// LS Electric XG5000 project: 2016-46
// PLC NewPLC
// module base 0 slot 0: 입출력 모듈:XBC-DR20E (DC 24V 입력 12점, 릴레이 출력 8점)

PROGRAM NewProgram (task: 스캔 프로그램)

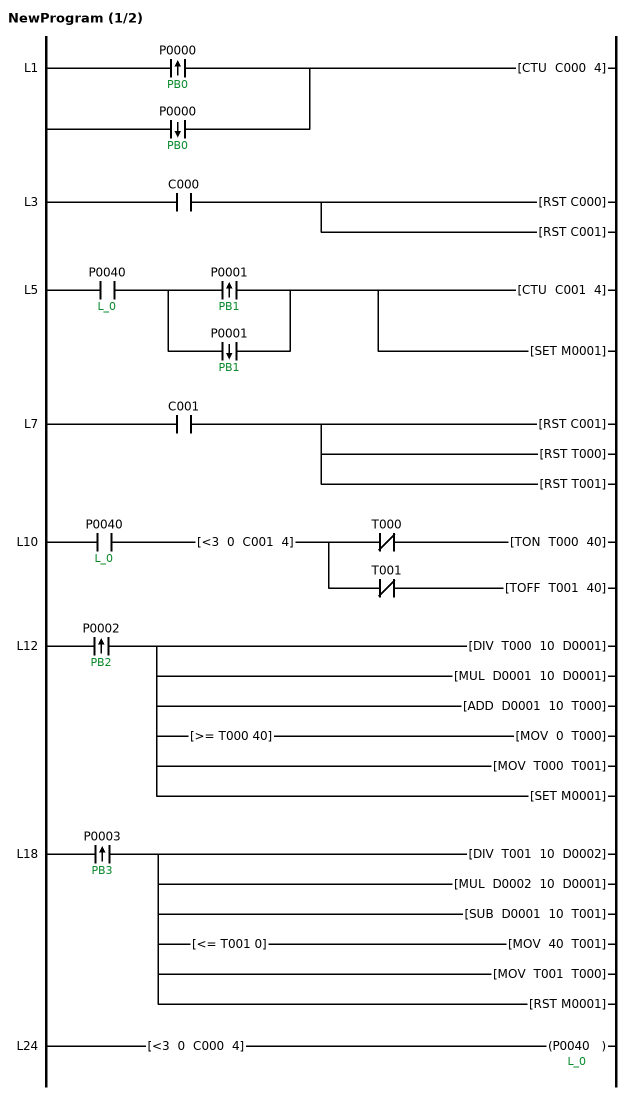
; L1
LOADP     P0000	// PB0
ORN       P0000	// PB0
CTU       C000 4
; L3
LOAD      C000
RST       C000
RST       C001
; L5
LOAD      P0040	// L_0
LOADP     P0001	// PB1
ORN       P0001	// PB1
AND LOAD
CTU       C001 4
SET       M0001
; L7
LOAD      C001
RST       C001
RST       T000
RST       T001
; L10
LOAD      P0040	// L_0
AND<3     0 C001 4
MPUSH
AND NOT   T000
TON       T000 40
MPOP
AND NOT   T001
TOFF      T001 40
; L12
LOADP     P0002	// PB2
DIV       T000 10 D0001
MUL       D0001 10 D0001
ADD       D0001 10 T000
MPUSH
AND>=     T000 40
MOV       0 T000
MPOP
MOV       T000 T001
SET       M0001
; L18
LOADP     P0003	// PB3
DIV       T001 10 D0002
MUL       D0002 10 D0001
SUB       D0001 10 T001
MPUSH
AND<=     T001 0
MOV       40 T001
MPOP
MOV       T001 T000
RST       M0001
; L24
LOAD<3    0 C000 4
OUT       P0040	// L_0

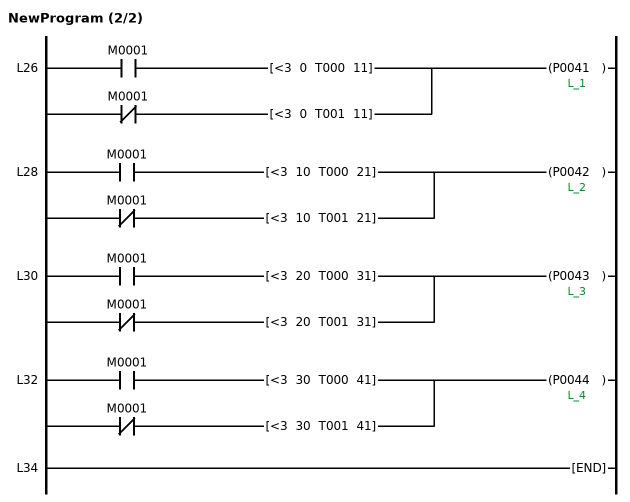
; L26
LOAD      M0001
AND<3     0 T000 11
LOAD NOT  M0001
AND<3     0 T001 11
OR LOAD
OUT       P0041	// L_1
; L28
LOAD      M0001
AND<3     10 T000 21
LOAD NOT  M0001
AND<3     10 T001 21
OR LOAD
OUT       P0042	// L_2
; L30
LOAD      M0001
AND<3     20 T000 31
LOAD NOT  M0001
AND<3     20 T001 31
OR LOAD
OUT       P0043	// L_3
; L32
LOAD      M0001
AND<3     30 T000 41
LOAD NOT  M0001
AND<3     30 T001 41
OR LOAD
OUT       P0044	// L_4
; L34
END